PROGRAM MAIN
VAR
END_VAR

END_PROGRAM

(* stored: Version 1.1.0.1
   POU MAIN: Id {ce101b60-7379-4d09-bc5d-d3755e26445e} *)
